FUNCTION_BLOCK FB_SaMElementResseting EXTENDS FB_SaMElement
VAR
END_VAR

METHOD FB_init : BOOL
VAR_INPUT
	bInitRetains : BOOL; // if TRUE, the retain variables are initialized (warm start / cold start)
	bInCopyCode : BOOL;  // if TRUE, the instance afterwards gets moved into the copy code (online change)
END_VAR
THIS^.SetText (eLocation := E_BaseLocation.pl, wsDescription := "Bazowanie");
THIS^.SetText (eLocation := E_BaseLocation.en, wsDescription := "Resetting");
THIS^.SetText (eLocation := E_BaseLocation.de, wsDescription := "Zurücksetzen");
THIS^.SetName (stName := THIS^.GetTexts ());
END_METHOD

METHOD PUBLIC InvokeStateForTopElement : BOOL
VAR_INPUT
	itfTopElement		: ITF_BaseSaMStateMethod;
END_VAR
InvokeStateForTopElement	:= itfTopElement.SP_Resetting ();
END_METHOD

END_FUNCTION_BLOCK

(* stored: Version 1.1.0.1
   POU FB_SaMElementResseting: Id {67aead33-83d6-0ab7-3f8b-522a487d85a7}, SpecialFunc None
   Method FB_init: Id {6fff04b8-dc37-07bc-2c4a-7f51181fe0fa}
   Method InvokeStateForTopElement: Id {2ee602f3-78d2-0112-3e31-a8892b806127} *)
